{attribute 'linkalways'} 
{attribute 'no_explicit_call' := 'This FB is a CLASS and must be accessed using methods or properties'}
{attribute 'enable_dynamic_creation'}
FUNCTION_BLOCK _ETcVnEdgeDetectionAlgorithm EXTENDS EnumDatatypeBase
VAR
	localData : ETcVnEdgeDetectionAlgorithm;
	activeData : REFERENCE TO ETcVnEdgeDetectionAlgorithm;
	enumBaseDatatype : _DINT(localData);
END_VAR

METHOD PRIVATE AddLocalEnumeration
VAR_INPUT
	Enumeration : T_MAXSTRING;
	Value : ETcVnEdgeDetectionAlgorithm;
END_VAR
AddEnumeration(Enumeration, Value);
END_METHOD

PROPERTY PUBLIC Address : PVOID
GET
Address := ADR(activeData);
END_GET
END_PROPERTY

METHOD PUBLIC ClearReference
VAR_INPUT
END_VAR
activeData REF= localData;
SetBaseDatatypeReference();
END_METHOD

METHOD PUBLIC Clone : I_Datatype
VAR
    pClone : POINTER TO _ETcVnEdgeDetectionAlgorithm;
END_VAR
pClone := __NEW(_ETcVnEdgeDetectionAlgorithm(InitialValue := Value));
Clone := pClone^;
END_METHOD

METHOD FB_init : BOOL
VAR_INPUT
	bInitRetains : BOOL; // if TRUE, the retain variables are initialized (warm start / cold start)
	bInCopyCode : BOOL;  // if TRUE, the instance afterwards gets moved into the copy code (online change)
	InitialValue : ETcVnEdgeDetectionAlgorithm;
END_VAR
localData := InitialValue;
AddBaseDatatype(enumBaseDatatype);
ClearReference();

AddLocalEnumeration('TCVN_EDA_INTERPOLATION', ETcVnEdgeDetectionAlgorithm.TCVN_EDA_INTERPOLATION);
AddLocalEnumeration('TCVN_EDA_APPROX_ERF', ETcVnEdgeDetectionAlgorithm.TCVN_EDA_APPROX_ERF);
AddLocalEnumeration('TCVN_EDA_APPROX_GAUSSIAN', ETcVnEdgeDetectionAlgorithm.TCVN_EDA_APPROX_GAUSSIAN);
END_METHOD

PROPERTY PUBLIC Identifier : T_MAXSTRING
GET
Identifier := 'ETcVnEdgeDetectionAlgorithm';
END_GET
END_PROPERTY

METHOD IsEnumeratorValueEqual : BOOL
VAR_INPUT
	Enumerator : I_KeyValueForwardEnumerator;
END_VAR
VAR
	storedValue : ETcVnEdgeDetectionAlgorithm;
END_VAR
IF NOT Enumerator.TryGet(storedValue) THEN
	RETURN;
END_IF

IsEnumeratorValueEqual := storedValue = activeData;
END_METHOD

METHOD PUBLIC MakeReferenceTo
VAR_INPUT
	ReferenceTarget : REFERENCE TO ETcVnEdgeDetectionAlgorithm;
END_VAR
activeData REF= ReferenceTarget;
SetBaseDatatypeReference();
END_METHOD

METHOD PROTECTED SetBaseDatatypeReference
VAR_INPUT
END_VAR
enumBaseDatatype.MakeReferenceTo(activeData);
END_METHOD

PROPERTY PUBLIC Size : UDINT
GET
Size := SIZEOF(activeData);
END_GET
END_PROPERTY

METHOD TryMakeReferenceTo : BOOL
VAR_INPUT
	Target : I_Datatype;
END_VAR
VAR
	targetAsEnum : I_EnumDatatype;
	pTargetData : POINTER TO ETcVnEdgeDetectionAlgorithm;
END_VAR
IF NOT Target.TryResolveAsEnumDatatype(targetAsEnum) THEN
	RETURN;
END_IF

IF targetAsEnum.Identifier <> Identifier THEN
	RETURN;
END_IF

pTargetData := Target.Address;
activeData REF= pTargetData^;
SetBaseDatatypeReference();
TryMakeReferenceTo := TRUE;
END_METHOD

PROPERTY PUBLIC Value : ETcVnEdgeDetectionAlgorithm
GET
Value := activeData;
END_GET
SET
activeData := Value;
END_SET
END_PROPERTY

END_FUNCTION_BLOCK

(* stored: Version 1.1.0.1, ProductVersion 3.1.4024.12
   POU _ETcVnEdgeDetectionAlgorithm: Id {443819f7-6384-46d2-b0dd-b12a9d90fd33}, SpecialFunc None
   Folder Constructor: Id {8c37c88e-f41e-4c74-9728-86fc8ef5bc7d}
   Folder Private: Id {609dbb72-e565-4282-af0b-cabbca980b2c}
   Folder Protected: Id {1bfc13ab-de53-467a-926d-c2a1ce7dd664}
   Method AddLocalEnumeration: Id {5d8b43e6-fddd-4a0d-9bbb-dcf8b76d768a}
   Property Address: Id {671a17c4-278c-49de-ac99-24d0f8fe310e}
   Get Get: Id {06a971d0-0bae-4b15-9d3b-ed1c1e603665}
   Method ClearReference: Id {7fffa638-fd5a-43ac-bed0-0decac5e15b2}
   Method Clone: Id {09d7f724-cb46-4d03-9a31-80b395463fa3}
   Method FB_init: Id {d39764e2-ef10-4fe6-909f-301c8737291e}
   Property Identifier: Id {e9cb8fba-982b-46a5-9d12-b2d108d74cb0}
   Get Get: Id {b99a8042-43af-4e1a-beea-825d15b6dcb4}
   Method IsEnumeratorValueEqual: Id {8fab751c-a665-41f0-bb37-acb32acf3b09}
   Method MakeReferenceTo: Id {0c136848-01c1-4fde-9b73-4683ffefc1ba}
   Method SetBaseDatatypeReference: Id {aed1aec0-19f0-44a1-bca4-5641dd29091e}
   Property Size: Id {40a9d66c-43bb-438e-bb52-aa43002c98bf}
   Get Get: Id {3443f9da-1bb1-4c0f-b151-2d635699f8c7}
   Method TryMakeReferenceTo: Id {e114cd7a-edf8-41c5-b618-74ca1865bf09}
   Property Value: Id {0c17d6dd-be31-4e5d-afa8-376d2d1a237d}
   Get Get: Id {2101839a-715c-4c82-8a00-c25762865d97}
   Set Set: Id {92e5dde7-38de-4e31-aecc-938c4613139b} *)
